{attribute 'linkalways'} 
{attribute 'no_explicit_call' := 'This FB is a CLASS and must be accessed using methods or properties'}
{attribute 'enable_dynamic_creation'}
FUNCTION_BLOCK RpcSynchronousReply IMPLEMENTS I_RpcSynchronousReply, I_RpcSynchronousReplyReadyToSend
VAR
	serializer : I_Serializer;
	serializerToSend : I_Serializer := serializer;
	serverResponse : I_ServerResponse;
	responseBuilder : RpcSynchronousResponseBuilder;
END_VAR

METHOD PUBLIC Compose : I_RpcResponseBuilder
VAR_INPUT
END_VAR
ResetInternalSerializer();
responseBuilder.Initialize(Serializer, ServerResponse);
Compose := responseBuilder;
END_METHOD

METHOD FB_init : BOOL
VAR_INPUT
	bInitRetains : BOOL; // if TRUE, the retain variables are initialized (warm start / cold start)
	bInCopyCode : BOOL;  // if TRUE, the instance afterwards gets moved into the copy code (online change)
	ServerResponse : I_ServerResponse;
	Serializer : I_Serializer;
END_VAR
THIS^.serverResponse := ServerResponse;
THIS^.serializer := Serializer;
END_METHOD

METHOD PUBLIC GetSerializer : I_Serializer
VAR_INPUT
END_VAR
GetSerializer := serializer.Clone();
END_METHOD

METHOD PUBLIC RejectWithMessage
VAR_INPUT
	Message : T_MAXSTRING;
END_VAR
serverResponse.Error(Message);
END_METHOD

METHOD PRIVATE ResetInternalSerializer
VAR_INPUT
END_VAR
serializer.Reset();
serializerToSend := serializer;
END_METHOD

METHOD PUBLIC Send
VAR
	jsonSize : UDINT;
	pJsonString : POINTER TO STRING;
END_VAR
jsonSize := serializerToSend.GetSeralizedDataLength();

IF jsonSize = 0 THEN
	serverResponse.Success();
END_IF

pJsonString := __NEW(BYTE, jsonSize);

IF NOT serializerToSend.TryGetSerialziedData(pJsonString, jsonSize) THEN
	serverResponse.Error('RPC Handler unable to get serialized data');
	__DELETE(pJsonString);
	RETURN;
END_IF

serverResponse.SuccessWithPayload(pJsonString, jsonSize);
__DELETE(pJsonString);
END_METHOD

METHOD PUBLIC WithBase64 : I_RpcSynchronousReplyReadyToSend
VAR_INPUT
	pBytes : POINTER TO BYTE;
	nBytes : DINT;
END_VAR
ResetInternalSerializer();
serializer.AddBase64(pBytes, nBytes);
WithBase64 := THIS^;
END_METHOD

METHOD PUBLIC WithBool : I_RpcSynchronousReplyReadyToSend
VAR_INPUT
	Value : BOOL;
END_VAR
ResetInternalSerializer();
serializer.AddBool(Value);
WithBool := THIS^;
END_METHOD

METHOD PUBLIC WithBytesAsHex : I_RpcSynchronousReplyReadyToSend
VAR_INPUT
	pBytes : POINTER TO BYTE;
	nBytes : DINT;
END_VAR
ResetInternalSerializer();
serializer.AddBytesAsHex(pBytes, nBytes);
WithBytesAsHex := THIS^;
END_METHOD

METHOD PUBLIC WithDateTime : I_RpcSynchronousReplyReadyToSend
VAR_INPUT
	Value : DATE_AND_TIME;
END_VAR
ResetInternalSerializer();
serializer.AddDateTime(Value);
WithDateTime := THIS^;
END_METHOD

METHOD PUBLIC WithDcTime : I_RpcSynchronousReplyReadyToSend
VAR_INPUT
	Value : DCTIME;
END_VAR
ResetInternalSerializer();
serializer.AddDcTime(Value);
WithDcTime := THIS^;
END_METHOD

METHOD PUBLIC WithDint : I_RpcSynchronousReplyReadyToSend
VAR_INPUT
	Value : DINT;
END_VAR
ResetInternalSerializer();
serializer.AddDint(Value);
WithDint := THIS^;
END_METHOD

METHOD PUBLIC WithFileTime : I_RpcSynchronousReplyReadyToSend
VAR_INPUT
	Value : FILETIME;
END_VAR
ResetInternalSerializer();
serializer.AddFileTime(Value);
WithFileTime := THIS^;
END_METHOD

METHOD PUBLIC WithLint : I_RpcSynchronousReplyReadyToSend
VAR_INPUT
	Value : LINT;
END_VAR
ResetInternalSerializer();
serializer.AddLint(Value);
WithLint := THIS^;
END_METHOD

METHOD PUBLIC WithLreal : I_RpcSynchronousReplyReadyToSend
VAR_INPUT
	Value : LREAL;
END_VAR
ResetInternalSerializer();
serializer.AddLreal(Value);
WithLreal := THIS^;
END_METHOD

METHOD PUBLIC WithNull : I_RpcSynchronousReplyReadyToSend
VAR_INPUT
END_VAR
ResetInternalSerializer();
serializer.AddNull();
WithNull := THIS^;
END_METHOD

METHOD PUBLIC WithObject : I_RpcSynchronousReplyReadyToSend
VAR_INPUT
	Object : I_Serializable;
END_VAR
ResetInternalSerializer();
Object.SerializeWith(serializer);
WithObject := THIS^;
END_METHOD

METHOD PUBLIC WithReal : I_RpcSynchronousReplyReadyToSend
VAR_INPUT
	Value : REAL;
END_VAR
ResetInternalSerializer();
serializer.AddReal(Value);
WithReal := THIS^;
END_METHOD

METHOD PUBLIC WithSerializedData : I_RpcSynchronousReplyReadyToSend
VAR_INPUT
	Serializer : I_Serializer;
END_VAR
ResetInternalSerializer();

IF Serializer = 0 THEN
	WithSerializedData := THIS^;
	RETURN;
END_IF

serializerToSend := Serializer;
WithSerializedData := THIS^;
END_METHOD

METHOD PUBLIC WithString : I_RpcSynchronousReplyReadyToSend
VAR_INPUT
	Value : T_MAXSTRING;
END_VAR
ResetInternalSerializer();
serializer.AddString(Value);
WithString := THIS^;
END_METHOD

METHOD PUBLIC WithUdint : I_RpcSynchronousReplyReadyToSend
VAR_INPUT
	Value : UDINT;
END_VAR
ResetInternalSerializer();
serializer.AddUdint(Value);
WithUdint := THIS^;
END_METHOD

METHOD PUBLIC WithUlint : I_RpcSynchronousReplyReadyToSend
VAR_INPUT
	Value : ULINT;
END_VAR
ResetInternalSerializer();
serializer.AddUlint(Value);
WithUlint := THIS^;
END_METHOD

END_FUNCTION_BLOCK

(* stored: Version 1.1.0.1, ProductVersion 3.1.4024.12
   POU RpcSynchronousReply: Id {c724498f-baf7-4f00-9137-6c3a66aa5cd0}, SpecialFunc None
   Folder Constructor: Id {12740898-8cc4-4e25-8ce9-9fc0666115c8}
   Folder Private: Id {dcb37f09-2ecb-4483-9579-8dcbc7918f05}
   Method Compose: Id {f36e2d3c-b4e8-439c-bf12-f5c1727b06af}
   Method FB_init: Id {58740322-7d24-44d6-95e0-bd81b1ebde4a}
   Method GetSerializer: Id {3c95a31f-9472-4fa2-8b38-a78edbb5c949}
   Method RejectWithMessage: Id {d016a36c-5bb1-48bd-ab36-b1534a482e0e}
   Method ResetInternalSerializer: Id {7aca96e4-a030-49b9-bab1-5f41b8d5633b}
   Method Send: Id {10656fd7-dd8c-4e2c-a443-082c5750c598}
   Method WithBase64: Id {1852c73b-7584-42d8-8595-d755b4b78f03}
   Method WithBool: Id {7e7403d7-f4cb-400d-8ab9-ff3aedbf57b4}
   Method WithBytesAsHex: Id {93903bbf-3c38-4980-8b1f-e2263cdb86e0}
   Method WithDateTime: Id {20014026-b2b6-43a2-93d7-0a69b7b874c8}
   Method WithDcTime: Id {601da881-ce92-48c2-b16a-901c433dac2e}
   Method WithDint: Id {38773dc1-5afc-4fbe-8d85-19dcb6f6dec0}
   Method WithFileTime: Id {ce3c3570-3dbd-429b-a0df-6122eef0b941}
   Method WithLint: Id {15fb45be-f8cd-476e-936e-95dd739d2ad8}
   Method WithLreal: Id {a6f94923-7cc9-4772-9c0b-daa067666dd8}
   Method WithNull: Id {a26a3275-f5d8-4d82-a9fa-28465a681661}
   Method WithObject: Id {8c148a58-c3ff-4c45-bfcd-db6bebceaad0}
   Method WithReal: Id {c45e6c4a-0553-4bd2-a3cd-0a5b5bd48d1b}
   Method WithSerializedData: Id {696c87ea-442f-4e8d-82ee-e793578eb606}
   Method WithString: Id {abf0072f-fd49-4976-9966-a04a5b803fee}
   Method WithUdint: Id {859ce20a-da2e-47f5-ba72-c20e7d8c636d}
   Method WithUlint: Id {c6871ed5-3419-4e00-9dd1-9901890cf472} *)
